FUNCTION_BLOCK FB_FixedPump IMPLEMENTS I_Pump


VAR CONSTANT
	fFlowRate : REAL := 20 ;
END_VAR
VAR
	bRunning : BOOL;
	fTotalVolume : REAL;
END_VAR

IF bRunning THEN
	fTotalVolume := fTotalVolume + fFlowRate;
END_IF

{warning 'add method implementation '}
METHOD GetFlowRate : REAL
GetFlowRate := fFlowRate;
END_METHOD

{warning 'add method implementation '}
METHOD GetTotalVolume : REAL
GetTotalVolume := fTotalVolume;
END_METHOD

{warning 'add method implementation '}
METHOD Start : BOOL
Start := bRunning := TRUE;
END_METHOD

{warning 'add method implementation '}
METHOD Stop : BOOL
bRunning := FALSE;
Stop := TRUE;
END_METHOD

END_FUNCTION_BLOCK

(* stored: Version 1.1.0.1, ProductVersion 3.1.4024.16
   POU FB_FixedPump: Id {85a93fcf-3d13-4ff8-a0e3-f9d7a51e2b47}, SpecialFunc None
   Method GetFlowRate: Id {a49ae1ce-71c1-4449-acd6-3dee743a172d}
   Method GetTotalVolume: Id {3aa09673-e930-42b8-b918-48a9fc96d79a}
   Method Start: Id {d8736705-b9f5-4ed1-bddd-ca7a242cf35c}
   Method Stop: Id {39ebd0e1-19e9-4be9-bae3-fe7a8cc9232b} *)
